{library PUBLIC}
TYPE DEVICE_TYPE :
(
	TYPE_ERROR:=-1, TYPE_SIMULATED:=0,  TYPE_ABB_1:=1, TYPE_GANTRY_1:=2
);
END_TYPE
//  TYPE_ERROR = '-1'

(* stored: Version 1.1.0.1, ProductVersion 3.1.4022.12
   EnumerationTextList DEVICE_TYPE: Id {78e8076b-e88f-46d2-a8e2-9bc517667895} *)
